// TIA Portal V15 export
// export: Created 2018-12-10T18:36:39.171501Z, ExportSetting WithDefaults, WithReadOnly, DisplayName Totally Integrated Automation Portal, DisplayVersion V15 Update 2, DisplayName TIA Portal Openness, DisplayVersion V15 Update 2, DisplayName STEP 7 Professional, DisplayVersion V15 Update 2, DisplayName STEP 7 Safety, DisplayVersion V15, DisplayName WinCC Professional, DisplayVersion V15 Update 2, DisplayName SIMATIC Visualization Architect, DisplayVersion V15 Update 1
DATA_BLOCK "FGDB_ROBNAME"   // DB94
TITLE = Robot Kuka KRC4
{ S7_Optimized_Access := 'FALSE' }
AUTHOR : integra
FAMILY : BS
VERSION : 0.5
// stored: AutoNumber true, CodeModifiedDate 2018-01-29T16:41:28.3431496Z, CompileDate 2018-02-20T10:24:35.9549134Z, CreationDate 2016-12-16T08:19:31.408454Z, DBAccessibleFromOPCUA true, InstanceOfName iFG_ROBOT, InstanceOfNumber 13, InstanceOfType FB, InterfaceModifiedDate 2018-01-24T13:15:23.6154787Z, IsConsistent true, IsKnowHowProtected false, ModifiedDate 2018-01-29T16:41:28.3431496Z, ParameterModified 2018-01-24T13:15:23.6154787Z, StructureModified 2018-01-24T13:15:23.6154787Z, UDAEnableTagReadback false
"iFG_ROBOT"
   // VAR_INPUT
   //    fct : Int;
   //    safetyStop : Bool;
   //    enableOut : Bool;
   //    autoStart : Bool;
   //    robotStop : Bool;
   //    ghostMode : Bool;
   //    reqSpecialPos : Bool;
   //    shutdownActivate : Bool;
   //    shutdownDeactivate : Bool;
   //    brakecheckPGNO : Int;
   //    referencePGNO : Int;
   // END_VAR
   // VAR_OUTPUT
   //    robotSelected : Bool;
   //    initialPosition : Bool;
   //    automaticOFF : Bool;
   //    readyPGNO_REQ : Bool;
   //    stop : Bool;
   //    specialPos : Bool;
   //    reqBrakecheck : Bool;
   //    reqReference : Bool;
   //    activeProgram : Int;
   //    shutdownActivated : Bool;
   //    shutdownDeactivated : Bool;
   //    Out_PO : "iUDT_PO_ROBOT";
   //    fault : Bool;
   //    faultExt : Bool;
   // END_VAR
   // VAR_IN_OUT
   //    In_PI : "iUDT_PI_ROBOT";
   //    selectionPGNO : Int;
   // END_VAR
   // VAR RETAIN
   //    idx : Int;
   //    sectionNumber : Int;
   //    deskNumber : Int;
   //    stationNumber : Int;
   //    dbNumber : Int;
   //    function : Int;
   //    numberInternalMessages : Int;
   //    numberExternalMessages : Int;
   //    PI_HMI : "iUDT_PI_ROBOT";
   //    F : Struct
   //       PLC_SUB : Bool;
   //       Prog_Start : Bool;
   //       SAK : Bool;
   //       fct : Bool;
   //       reqGhost : Bool;
   //       drivesOn : Bool;
   //       ROBOT_fault : Bool;
   //       DFE : Bool;
   //       reference : Bool;
   //       brakeCheck : Bool;
   //       peripheralINPUT : Bool;
   //       brakeReachedLimit : Bool;
   //       acyclicServiceRobot : Bool;
   //       robotStopped : Bool;
   //       energyLockout : Bool;
   //       energySwitchingOn : Bool;
   //       acyclicServicePLC : Bool;
   //       acyclicData : Bool;
   //    END_STRUCT;
   //    W : Struct
   //       robotDeselected : Bool;
   //       noAutomatic : Bool;
   //       brakeCheck : Bool;
   //       override : Bool;
   //    END_STRUCT;
   //    Masks : Struct
   //       disableFault1_8 : Byte;
   //       disableFault9_16 : Byte;
   //       prodRelevantFault1_8 : Byte;
   //       prodRelevantFault9_16 : Byte;
   //       prodRelevantWarningt_1_8 : Byte;
   //    END_STRUCT;
   //    LastState : Struct
   //       fault_1_8 : Byte;
   //       fault_9_16 : Byte;
   //       warning_1_8 : Byte;
   //    END_STRUCT;
   //    IfcFGExternal : "iUDT_IFC_SYS_EXTERNAL_ALARM";
   //    Tmr : Struct
   //       s_1 { S7_SetPoint := 'True'} : Int;
   //       a_1 : Int;
   //       s_2 { S7_SetPoint := 'True'} : Int;
   //       a_2 : Int;
   //       s_3 { S7_SetPoint := 'True'} : Int;
   //       a_3 : Int;
   //       s_4 { S7_SetPoint := 'True'} : Int;
   //       a_4 : Int;
   //       s_5 { S7_SetPoint := 'True'} : Int;
   //       a_5 : Int;
   //       s_6 { S7_SetPoint := 'True'} : Int;
   //       a_6 : Int;
   //       s_7 { S7_SetPoint := 'True'} : Int;
   //       a_7 : Int;
   //       s_8 { S7_SetPoint := 'True'} : Int;
   //       a_8 : Int;
   //       s_9 { S7_SetPoint := 'True'} : Int;
   //       a_9 : Int;
   //       s_10 { S7_SetPoint := 'True'} : Int;
   //       a_10 : Int;
   //    END_STRUCT;
   //    ExtP : Struct
   //       setup : Bool;
   //       auto : Bool;
   //       enIn : Bool;
   //       ack : Bool;
   //    END_STRUCT;
   //    StM : Struct
   //       fault : Bool;
   //       setup : Bool;
   //       auto : Bool;
   //       warning : Bool;
   //       eStop : Bool;
   //       safetyStop : Bool;
   //       enableIn : Bool;
   //       enableOutForward : Bool;
   //       enableOutBackward : Bool;
   //       faultPr : Bool;
   //       pairMon : Bool;
   //       specialMode : Bool;
   //       "13" : Bool;
   //       "14" : Bool;
   //       "15" : Bool;
   //       "16" : Bool;
   //       "17" : Bool;
   //       "18" : Bool;
   //       "19" : Bool;
   //       "20" : Bool;
   //       "21" : Bool;
   //       "22" : Bool;
   //       "23" : Bool;
   //       "24" : Bool;
   //       "25" : Bool;
   //       "26" : Bool;
   //       "27" : Bool;
   //       "28" : Bool;
   //       "29" : Bool;
   //       "30" : Bool;
   //       "31" : Bool;
   //       "32" : Bool;
   //    END_STRUCT;
   //    VB : Struct
   //       safeRobot : Bool;
   //       robotInitalState : Bool;
   //       robotProgromSelection : Bool;
   //       robotStart : Bool;
   //       robotRunning : Bool;
   //       "6" : Bool;
   //       "7" : Bool;
   //       "8" : Bool;
   //       "9" : Bool;
   //       "10" : Bool;
   //       "11" : Bool;
   //       "12" : Bool;
   //       "13" : Bool;
   //       "14" : Bool;
   //       "15" : Bool;
   //       "16" : Bool;
   //       "17" : Bool;
   //       "18" : Bool;
   //       "19" : Bool;
   //       "20" : Bool;
   //       "21" : Bool;
   //       "22" : Bool;
   //       "23" : Bool;
   //       "24" : Bool;
   //       "25" : Bool;
   //       "26" : Bool;
   //       "27" : Bool;
   //       "28" : Bool;
   //       "29" : Bool;
   //       "30" : Bool;
   //       "31" : Bool;
   //       "32" : Bool;
   //    END_STRUCT;
   //    VCB : Struct
   //       ack : Bool;
   //       readActivationCode : Bool;
   //       storedActivationCode : Bool;
   //    END_STRUCT;
   //    TmrB : Struct
   //       "1_Enable" : Bool;
   //       "1_Run" : Bool;
   //       "1_Done" : Bool;
   //       "2_Enable" : Bool;
   //       "2_Run" : Bool;
   //       "2_Done" : Bool;
   //       "3_Enable" : Bool;
   //       "3_Run" : Bool;
   //       "3_Done" : Bool;
   //       "4_Enable" : Bool;
   //       "4_Run" : Bool;
   //       "4_Done" : Bool;
   //       "5_Enable" : Bool;
   //       "5_Run" : Bool;
   //       "5_Done" : Bool;
   //       "6_Enable" : Bool;
   //       "6_Run" : Bool;
   //       "6_Done" : Bool;
   //       "7_Enable" : Bool;
   //       "7_Run" : Bool;
   //       "7_Done" : Bool;
   //       "8_Enable" : Bool;
   //       "8_Run" : Bool;
   //       "8_Done" : Bool;
   //       "9_Enable" : Bool;
   //       "9_Run" : Bool;
   //       "9_Done" : Bool;
   //       "10_Enable" : Bool;
   //       "10_Run" : Bool;
   //       "10_Done" : Bool;
   //    END_STRUCT;
   //    D : Struct
   //       visuAck : Bool;
   //       enableIn : Bool;
   //       withRobot : Bool := true;
   //       changeMode : Bool;
   //       programToNEAR_POSRET : Bool;
   //       releaseROBOTerror : Bool;
   //       auxDelayROBOTerror : Bool;
   //       delayROBOTerror : Bool;
   //       startAfterSTOPMESS : Bool;
   //       fPSTOPMESS : Bool;
   //       delayedMoveEnable : Bool;
   //       fPLiveBitRobot : Bool;
   //       auxDelayedMoveEnable : Bool;
   //       externalStart : Bool;
   //       fPForRestart : Bool;
   //       fPNEARPOSRET : Bool;
   //       programAct : Bool;
   //       delayGhostMode : Bool;
   //       reqBrakecheck : Bool;
   //       reqMasteringcheck : Bool;
   //       DRIVES_ON : Bool;
   //       MOVE_ENABLE : Bool;
   //       CONF_MESS : Bool;
   //       PGNO_VALID : Bool;
   //       PGNO_PARITY : Bool;
   //       ANFSP : Bool;
   //       GBA : Bool;
   //       GBNA : Bool;
   //       acyclicDataDone : Bool;
   //       fPacyclicDataDone : Bool;
   //       fNacyclicDataRecv : Bool;
   //       initialPosition : Bool;
   //       readActivationCode : Bool;
   //       shutdownActivated : Bool;
   //       shutdownDeactivated : Bool;
   //    END_STRUCT;
   //    V : Struct
   //       runtime : UInt;
   //       auxPGNO : Int;
   //       PGNO : Int;
   //       activePGNO : Int;
   //       ID_HW_IO_StandardModul : HW_IO;
   //       ID_HW_IO_SafetyModul : HW_IO;
   //       safetyActivationCodeCurrent : Array[1..4] of Byte;
   //       safetyActivationCodeStored : Array[1..4] of Byte;
   //       GEOADDR : GEOADDR;
   //    END_STRUCT;
   //    "RB-RB" : Struct
   //       R_I0361 : Bool;
   //       R_I0362 : Bool;
   //       R_I0363 : Bool;
   //       R_I0364 : Bool;
   //       R_I0365 : Bool;
   //       R_I0366 : Bool;
   //       R_I0367 : Bool;
   //       R_I0368 : Bool;
   //       R_I0369 : Bool;
   //       R_I0370 : Bool;
   //       R_I0371 : Bool;
   //       R_I0372 : Bool;
   //       R_I0373 : Bool;
   //       R_I0374 : Bool;
   //       R_I0375 : Bool;
   //       R_I0376 : Bool;
   //    END_STRUCT;
   //    IfcTECH : "iUDT_IFC_ROBOT_TECH";
   //    IfcAcyclic : "iIF_ROBOT_ACYCLICDATA";
   //    RDREC_Instance : RDREC;
   // END_VAR
BEGIN
END_DATA_BLOCK
